FUNCTION_BLOCK CollectionChangedEventHandler EXTENDS CollectionEventHandler

METHOD PUBLIC HandleEvent
VAR_INPUT
	Event : I_Event;
END_VAR
VAR
	changedEvent : I_CollectionChangedEvent;
END_VAR
IF __QUERYINTERFACE(Event, changedEvent) THEN
	_eventReceived := TRUE;
	fromExpected := changedEvent.Target = expectedOriginator;
END_IF
END_METHOD

END_FUNCTION_BLOCK

(* stored: Version 1.1.0.1, ProductVersion 3.1.4024.12
   POU CollectionChangedEventHandler: Id {df2f6f47-3554-0f60-2568-09df0fc3bcd5}, SpecialFunc None
   Method HandleEvent: Id {6bd60c70-efdd-053c-3ebf-6416aa65ac49} *)
